Fanuc KAREL source: kb00167.KL

-- PROVISIONAL review KL for V940-1; original PC SHA256 af862a1623bce90aaf267ebd17771eb059bf094190cff5854903d36524c733be
-- Incomplete behavior may be omitted. Consult companion uncertainty JSON. Do not deploy.
PROGRAM KB00167
%NOLOCKGROUP
BEGIN
  -- V9_ZERO_TABLE_METADATA_HINT layout=0002_ascii; no indexed target words; source/name/runtime held
  -- UNRESOLVED_PC offsets 5-12; opcodes 9D,23
  -- UNRESOLVED_PC offsets 17-24; opcodes 9D,23
  -- UNRESOLVED_PC offsets 29-36; opcodes 9D,23
  -- UNRESOLVED_PC offsets 41-77; opcodes 27,22,22,22,1C,22,27,9D,31
  -- UNRESOLVED_PC offsets 82-86; opcodes 7F
END KB00167
